(* PLC project Tc2_Coupler.stLibVersion_Tc2_Coupler Demo, tc3-libraries-kb TwinCAT 3.1 *)
(* stored: creationDateTime 2026-05-10T09:00:00, modificationDateTime 2026-05-10T09:00:00 *)

PROGRAM P_Demo_stLibVersion_Tc2_Coupler
  VAR
    stMyVer : ST_LibVersion;  (* 本地副本（监视用） *)
    bOk : BOOL;  (* 版本检查结果 *)
  END_VAR

            // ============================================================
// Tc2_Coupler.stLibVersion_Tc2_Coupler 演示程序
// ============================================================
// 注意：项目须引用 Tc2_Coupler 与 Tc2_System（ST_LibVersion / F_CmpLibVersion）
// 验证步骤：
//   1. 编译 + 登录
//   2. 在线监视 stMyVer.iMajor/iMinor/iBuild — 应显示 1.1.1
//   3. 在线监视 bOk — 应为 TRUE
// ============================================================

stMyVer := stLibVersion_Tc2_Coupler;

bOk := F_CmpLibVersion(
    stLibVersion := stLibVersion_Tc2_Coupler,
    iMajor       := 1,
    iMinor       := 1,
    iBuild       := 1,
    iRevision    := 0,
    nCmpType     := E_CmpLibVersion.GreaterOrEqual
);

          
END_PROGRAM
